// TIA Portal V17 export
// export: Created 2025-03-10T13:09:25.1133603Z, ExportSetting WithDefaults, DisplayName Totally Integrated Automation Portal, DisplayVersion V17 Update 8, DisplayName TIA Portal Openness, DisplayVersion V17 Update 8, DisplayName TIA Portal Version Control Interface, DisplayVersion V17, DisplayName SINAMICS Startdrive Advanced, DisplayVersion V17 SP2, DisplayName SINAMICS Startdrive G110M, G120, G120C, G120D, G120P, G115D, DisplayVersion V17 SP2, DisplayName SINAMICS Startdrive G130, G150, S120, S150, SINAMICS MV, S210, DisplayVersion V17 SP2, DisplayName STEP 7 Professional, DisplayVersion V17 Update 8, DisplayName SINUMERIK ONE STEP 7 Toolbox, DisplayVersion V17 Update 12, DisplayName SINUMERIK 840D sl STEP 7 Toolbox, DisplayVersion V17 Update 12, DisplayName STEP 7 Safety, DisplayVersion V17 Update 6, DisplayName WinCC Advanced, DisplayVersion V17 Update 8
DATA_BLOCK "LBP_PIServices"   // DB16
TITLE = PI Services / Servicios de IP / PI-Dienste
{ DB_Accessible_From_OPC_UA := 'FALSE' }
// Interface for LBP_ReqPIService [FB7], contains definitions for all available PI services. / Interfaz para LBP_ReqPIService [FB7], contiene definiciones para todos los servicios PI disponibles. / Schnittstelle für LBP_ReqPIService [FB7], enthält Definitionen für alle verfügbaren PI-Dienste.
// stored: DBAccessibleFromOPCUA false, DBAccessibleFromWebserver true, IsOnlyStoredInLoadMemory false, IsWriteProtectedInAS false
   VAR
      SELECT : Struct
         PIName : String[10] := '_N_SELECT';
         p01 : Byte := BYTE#16#03;   // Bereich/Einheit / Area / Unit / Área/unidad
         p02 : Char := '2';   // Bereichskennung / Area identifier / Identificador de área
         p11 : Byte := BYTE#16#FD;   // Pfad-Name / Path name / Nombre de ruta
         p12 : Byte := BYTE#16#13;   // String beliebig lang ungeradzahlig ergaenzen / Add string with arbitrary number of odd numbers / Completar string con cifras impares de una longitud cualquiera
         p21 : Byte := BYTE#16#FE;   // Programm-Name / Program name / Nombre de programa
         p22 : Byte := BYTE#16#13;   // String beliebig lang ungeradzahlig ergaenzen / Add string with arbitrary number of odd numbers / Completar string con cifras impares de una longitud cualquiera
      END_STRUCT;
      ASUP : Struct
         PIName : String[10] := '_N_ASUP__';
         p01 : Byte := BYTE#16#03;   // Bereich/Einheit / Area / Unit / Área/unidad
         p02 : Char := '2';   // Bereichskennung / Area identifier / Identificador de área
         p11 : Byte := BYTE#16#03;   // Interrupt-Nummer / Interrupt number / Número de interrupción
         p12 : Byte := BYTE#16#05;   // Int aus WORD-Spezifikation / Int from WORD specification / INT a partir de especificación WORD
         p21 : Byte := BYTE#16#03;   // Priorität / Priority / Prioridad
         p22 : Byte := BYTE#16#05;   // Int aus WORD-Spezifikation / Int from WORD specification / INT a partir de especificación WORD
         p31 : Byte := BYTE#16#01;   // Liftfast
         p32 : Byte := BYTE#16#05;   // Int aus WORD-Spezifikation / Int from WORD specification / INT a partir de especificación WORD
         p41 : Byte := BYTE#16#01;   // Blocksync / Sinc bloque
         p42 : Byte := BYTE#16#05;   // Int aus WORD-Spezifikation / Int from WORD specification / INT a partir de especificación WORD
         p51 : Byte := BYTE#16#FD;   // Pfad-Name / Path name / Nombre de ruta
         p52 : Byte := BYTE#16#13;   // String beliebig lang ungeradzahlig ergaenzen / Add string with arbitrary number of odd numbers / Completar string con cifras impares de una longitud cualquiera
         p61 : Byte := BYTE#16#FE;   // Programm-Name / Program name / Nombre de programa
         p62 : Byte := BYTE#16#13;   // String beliebig lang ungeradzahlig ergaenzen / Add string with arbitrary number of odd numbers / Completar string con cifras impares de una longitud cualquiera
      END_STRUCT;
      FINDBL : Struct
         PIName : String[10] := '_N_FINDBL';
         p01 : Byte := BYTE#16#03;   // Bereich/Einheit / Area / Unit / Área/unidad
         p02 : Char := '2';
         p11 : Byte := BYTE#16#01;   // Vorlaufmodus / Preprocessing mode / Modo de marcha previa
         p12 : Byte := BYTE#16#04;   // Word aus WORD-Spezifikation / Word from WORD specification / Word desde especificación WORD
      END_STRUCT;
      SETUFR : Struct
         PIName : String[10] := '_N_SETUFR';
         p01 : Byte := BYTE#16#03;   // Bereich/Einheit / Area / Unit / Área/unidad
         p02 : Char := '2';
      END_STRUCT;
      CANCEL : Struct
         PIName : String[10] := '_N_CANCEL';
         p01 : Byte := BYTE#16#03;   // Bereich/Einheit / Area / Unit / Área/unidad
         p02 : Char := '0';
      END_STRUCT;
      DELETO : Struct
         PIName : String[10] := '_N_DELETO';
         p01 : Byte := BYTE#16#03;   // Bereich/Einheit / Area / Unit / Área/unidad
         p02 : Char := '4';
         p11 : Byte := BYTE#16#05;   // T-Nummer / T number / N.º T
         p12 : Byte := BYTE#16#05;   // Int aus WORD-Spezifikation / Int from WORD specification / INT a partir de especificación WORD
      END_STRUCT;
      CREATO : Struct
         PIName : String[10] := '_N_CREATO';
         p01 : Byte := BYTE#16#03;   // Bereich/Einheit / Area / Unit / Área/unidad
         p02 : Char := '4';
         p11 : Byte := BYTE#16#05;   // T-Nummer / T number / N.º T
         p12 : Byte := BYTE#16#05;   // Int aus WORD-Spezifikation / Int from WORD specification / INT a partir de especificación WORD
      END_STRUCT;
      CREACE : Struct
         PIName : String[10] := '_N_CREACE';
         p01 : Byte := BYTE#16#03;   // Bereich/Einheit / Area / Unit / Área/unidad
         p02 : Char := '4';
         p11 : Byte := BYTE#16#05;   // T-Nummer / T number / N.º T
         p12 : Byte := BYTE#16#05;   // Int aus WORD-Spezifikation / Int from WORD specification / INT a partir de especificación WORD
      END_STRUCT;
      TMCRTO : Struct
         PIName : String[10] := '_N_TMCRTO';
         p01 : Byte := BYTE#16#03;   // Bereich/Einheit / Area / Unit / Área/unidad
         p02 : Char := '4';
         p11 : Byte := BYTE#16#20;   // Werkzeugkennung, Leerzeichen hinzufügen / Tool identifier, add blank / Identificador de herramienta, agregar espacio en blanco
         p12 : Byte := BYTE#16#13;   // Stringkennung! / String identifier! / ¡Identificador de string!
         p21 : Byte := BYTE#16#05;   // T-Nummer / T number / N.º T
         p22 : Byte := BYTE#16#05;   // Int aus WORD-Spezifikation / Int from WORD specification / INT a partir de especificación WORD
         p31 : Byte := BYTE#16#05;   // Duplo Nummer / Duplo number / Número duplo
         p32 : Byte := BYTE#16#05;   // Int aus WORD-Spezifikation / Int from WORD specification / INT a partir de especificación WORD
      END_STRUCT;
      TMFDPL : Struct
         PIName : String[10] := '_N_TMFDPL';
         p01 : Byte := BYTE#16#03;   // Bereich/Einheit / Area / Unit / Área/unidad
         p02 : Char := '4';
         p11 : Byte := BYTE#16#05;   // T-Nummer / T number / N.º T
         p12 : Byte := BYTE#16#05;   // Int aus WORD-Spezifikation / Int from WORD specification / INT a partir de especificación WORD
         p21 : Byte := BYTE#16#05;   // Platznummer (Ziel) / Location number (target) / Número de puesto (destino)
         p22 : Byte := BYTE#16#05;   // Int aus WORD-Spezifikation / Int from WORD specification / INT a partir de especificación WORD
         p31 : Byte := BYTE#16#05;   // Magazinnummer (Ziel) / Magazine number (target) / Número de almacén (destino)
         p32 : Byte := BYTE#16#05;   // Int aus WORD-Spezifikation / Int from WORD specification / INT a partir de especificación WORD
         p41 : Byte := BYTE#16#05;   // Platznummer (Bezug) / Location number (reference) / Número de puesto (referencia)
         p42 : Byte := BYTE#16#05;   // Int aus WORD-Spezifikation / Int from WORD specification / INT a partir de especificación WORD
         p51 : Byte := BYTE#16#05;   // Magazin-Nummer (Bezug) / Magazine number (reference) / Número de almacén (referencia)
         p52 : Byte := BYTE#16#05;   // Int aus WORD-Spezifikation / Int from WORD specification / INT a partir de especificación WORD
      END_STRUCT;
      TMMVTL : Struct
         PIName : String[10] := '_N_TMMVTL';
         p01 : Byte := BYTE#16#03;   // Bereich/Einheit / Area / Unit / Área/unidad
         p02 : Char := '4';
         p11 : Byte := BYTE#16#05;   // T-Nummer / T number / N.º T
         p12 : Byte := BYTE#16#05;   // Int aus WORD-Spezifikation / Int from WORD specification / INT a partir de especificación WORD
         p21 : Byte := BYTE#16#05;   // Platznummer (Quelle) / Location number (source) / Número de puesto (origen)
         p22 : Byte := BYTE#16#05;   // Int aus WORD-Spezifikation / Int from WORD specification / INT a partir de especificación WORD
         p31 : Byte := BYTE#16#05;   // Magazin-Nummer (Quelle) / Magazine number (source) / Número de almacén (origen)
         p32 : Byte := BYTE#16#05;   // Int aus WORD-Spezifikation / Int from WORD specification / INT a partir de especificación WORD
         p41 : Byte := BYTE#16#05;   // Platznummer (Ziel) / Location number (target) / Número de puesto (destino)
         p42 : Byte := BYTE#16#05;   // Int aus WORD-Spezifikation / Int from WORD specification / INT a partir de especificación WORD
         p51 : Byte := BYTE#16#05;   // Magazin-Nummer (Ziel) / Magazine number (target) / Número de almacén (destino)
         p52 : Byte := BYTE#16#05;   // Int aus WORD-Spezifikation / Int from WORD specification / INT a partir de especificación WORD
      END_STRUCT;
      TMPCIT : Struct
         PIName : String[10] := '_N_TMPCIT';
         p01 : Byte := BYTE#16#03;   // Bereich/Einheit / Area / Unit / Área/unidad
         p02 : Char := '4';
         p11 : Byte := BYTE#16#03;   // Spindelnummer / Spindle number / Número de cabezal
         p12 : Byte := BYTE#16#05;   // Int aus WORD-Spezifikation / Int from WORD specification / INT a partir de especificación WORD
         p21 : Byte := BYTE#16#05;   // Inkrement Wert / Increment value / Valor incremental
         p22 : Byte := BYTE#16#05;   // Int aus WORD-Spezifikation / Int from WORD specification / INT a partir de especificación WORD
      END_STRUCT;
      TMPOSM : Struct
         PIName : String[10] := '_N_TMPOSM';
         p01 : Byte := BYTE#16#03;   // Bereich/Einheit / Area / Unit / Área/unidad
         p02 : Char := '4';
         p11 : Byte := BYTE#16#05;   // T-Nummer / T number / N.º T
         p12 : Byte := BYTE#16#05;   // Int aus WORD-Spezifikation / Int from WORD specification / INT a partir de especificación WORD
         p21 : Byte := BYTE#16#20;   // Werkzeugbezeichner, Leerzeichen hinzufügen / Tool identifier, add blank / Identificador de herramienta, agregar espacio en blanco
         p22 : Byte := BYTE#16#13;   // Stringkennung! / String identifier! / ¡Identificador de string!
         p31 : Byte := BYTE#16#05;   // Duplo Nummer / Duplo number / Número duplo
         p32 : Byte := BYTE#16#05;   // Int aus WORD-Spezifikation / Int from WORD specification / INT a partir de especificación WORD
         p41 : Byte := BYTE#16#05;   // Platznummer (Quelle) / Location number (source) / Número de puesto (origen)
         p42 : Byte := BYTE#16#05;   // Int aus WORD-Spezifikation / Int from WORD specification / INT a partir de especificación WORD
         p51 : Byte := BYTE#16#05;   // Magazin-Nummer (Quelle) / Magazine number (source) / Número de almacén (origen)
         p52 : Byte := BYTE#16#05;   // Int aus WORD-Spezifikation / Int from WORD specification / INT a partir de especificación WORD
         p61 : Byte := BYTE#16#05;   // Platznummer (Ziel) / Location number (target) / Número de puesto (destino)
         p62 : Byte := BYTE#16#05;   // Int aus WORD-Spezifikation / Int from WORD specification / INT a partir de especificación WORD
         p71 : Byte := BYTE#16#05;   // Magazin-Nummer (Ziel) / Magazine number (target) / Número de almacén (destino)
         p72 : Byte := BYTE#16#05;   // Int aus WORD-Spezifikation / Int from WORD specification / INT a partir de especificación WORD
      END_STRUCT;
      DIGION : Struct
         PIName : String[10] := '_N_DIGION';
         p01 : Byte := BYTE#16#03;   // Bereich/Einheit / Area / Unit / Área/unidad
         p02 : Char := '2';
      END_STRUCT;
      DIGIOF : Struct
         PIName : String[10] := '_N_DIGIOF';
         p01 : Byte := BYTE#16#03;   // Bereich/Einheit / Area / Unit / Área/unidad
         p02 : Char := '2';
      END_STRUCT;
      CONFIG : Struct
         PIName : String[10] := '_N_CONFIG';
         p01 : Byte := BYTE#16#03;   // Bereich/Einheit / Area / Unit / Área/unidad
         p02 : Char := '0';
         p11 : Byte := BYTE#16#02;   // Klassifizierung / Classification / Clasificación
         p12 : Byte := BYTE#16#04;   // Int aus WORD-Spezifikation / Int from WORD specification / INT a partir de especificación WORD
      END_STRUCT;
      LOGIN : Struct
         PIName : String[10] := '_N_LOGIN_';
         p01 : Byte := BYTE#16#03;   // Bereich/Einheit / Area / Unit / Área/unidad
         p02 : Char := '0';
         p11 : Byte := BYTE#16#20;   // Kennwort (8 - 32 Zeichen) / Password (8 to 32 characters) / Contraseña (de 8 a 32 caracteres)
         p12 : Byte := BYTE#16#13;   // Stringkennung! / String identifier! / ¡Identificador de string!
      END_STRUCT;
      LOGOUT : Struct
         PIName : String[10] := '_N_LOGOUT';
         p01 : Byte := BYTE#16#03;   // Bereich/Einheit / Area / Unit / Área/unidad
         p02 : Char := '0';
      END_STRUCT;
      MMCSEM : Struct
         PIName : String[10] := '_N_MMCSEM';
         p01 : Byte := BYTE#16#03;   // Bereich/Einheit / Area / Unit / Área/unidad
         p02 : Char := '2';
         p11 : Byte := BYTE#16#03;   // Funktionsnummer / Function number / Número de función
         p12 : Byte := BYTE#16#05;   // Int aus WORD-Spezifikation / Int from WORD specification / INT a partir de especificación WORD
         p21 : Byte := BYTE#16#01;   // Semaphore-Wert / Semaphore value / Valor de semáforo
         p22 : Byte := BYTE#16#05;   // Int aus WORD-Spezifikation / Int from WORD specification / INT a partir de especificación WORD
      END_STRUCT;
      DELECE : Struct
         PIName : String[10] := '_N_DELECE';
         p01 : Byte := BYTE#16#03;   // Bereich/Einheit / Area / Unit / Área/unidad
         p02 : Char := '4';
         p11 : Byte := BYTE#16#05;   // T-Nummer / T number / N.º T
         p12 : Byte := BYTE#16#05;   // Int aus WORD-Spezifikation / Int from WORD specification / INT a partir de especificación WORD
         p21 : Byte := BYTE#16#05;   // D-Nummer / D number / N.º D
         p22 : Byte := BYTE#16#05;   // Int aus WORD-Spezifikation / Int from WORD specification / INT a partir de especificación WORD
      END_STRUCT;
      CRCEDN : Struct
         PIName : String[10] := '_N_CRCEDN';
         p01 : Byte := BYTE#16#03;   // Bereich/Einheit / Area / Unit / Área/unidad
         p02 : Char := '4';
         p11 : Byte := BYTE#16#05;   // T-Nummer / T number / N.º T
         p12 : Byte := BYTE#16#05;   // Int aus WORD-Spezifikation / Int from WORD specification / INT a partir de especificación WORD
         p21 : Byte := BYTE#16#05;   // D-Nummer / D number / N.º D
         p22 : Byte := BYTE#16#05;   // Int aus WORD-Spezifikation / Int from WORD specification / INT a partir de especificación WORD
      END_STRUCT;
      TSEARC : Struct
         PIName : String[10] := '_N_TSEARC';
         p01 : Byte := BYTE#16#03;   // Bereich/Einheit / Area / Unit / Área/unidad
         p02 : Char := '4';
         p11 : Byte := BYTE#16#05;   // von: Magazin-Nummer / from: Magazine number / desde: número de almacén
         p12 : Byte := BYTE#16#05;   // Int aus WORD-Spezifikation / Int from WORD specification / INT a partir de especificación WORD
         p21 : Byte := BYTE#16#05;   // von: Platznummer / from: Location number / desde: número de puesto
         p22 : Byte := BYTE#16#05;   // Int aus WORD-Spezifikation / Int from WORD specification / INT a partir de especificación WORD
         p31 : Byte := BYTE#16#05;   // bis: Magazin-Nummer / up to: Magazine number / hasta: número de almacén
         p32 : Byte := BYTE#16#05;   // Int aus WORD-Spezifikation / Int from WORD specification / INT a partir de especificación WORD
         p41 : Byte := BYTE#16#05;   // bis: Platznummer / up to: Location number / hasta: número de puesto
         p42 : Byte := BYTE#16#05;   // Int aus WORD-Spezifikation / Int from WORD specification / INT a partir de especificación WORD
         p51 : Byte := BYTE#16#05;   // Nummer des Referenz-Magazins / Number of reference magazine / Número del almacén de referencia
         p52 : Byte := BYTE#16#05;   // Int aus WORD-Spezifikation / Int from WORD specification / INT a partir de especificación WORD
         p61 : Byte := BYTE#16#05;   // Nummer des Referenz-Platzes / Number of reference location / Número del puesto de referencia
         p62 : Byte := BYTE#16#05;   // Int aus WORD-Spezifikation / Int from WORD specification / INT a partir de especificación WORD
         p71 : Byte := BYTE#16#01;   // Suchrichtung / Search direction / Sentido de búsqueda
         p72 : Byte := BYTE#16#05;   // Int aus WORD-Spezifikation / Int from WORD specification / INT a partir de especificación WORD
         p81 : Byte := BYTE#16#01;   // Eigenschaften der Werkzeuge / Tool properties / Propiedades de las herramientas
         p82 : Byte := BYTE#16#05;   // Int aus WORD-Spezifikation / Int from WORD specification / INT a partir de especificación WORD
      END_STRUCT;
      TMFPBP : Struct
         PIName : String[10] := '_N_TMFPBP';
         p01 : Byte := BYTE#16#03;   // Bereich/Einheit / Area / Unit / Área/unidad
         p02 : Char := '4';
         p11 : Byte := BYTE#16#05;   // von: Magazin-Nummer / from: Magazine number / desde: número de almacén
         p12 : Byte := BYTE#16#05;   // Int aus WORD-Spezifikation / Int from WORD specification / INT a partir de especificación WORD
         p21 : Byte := BYTE#16#05;   // von: Platznummer / from: Location number / desde: número de puesto
         p22 : Byte := BYTE#16#05;   // Int aus WORD-Spezifikation / Int from WORD specification / INT a partir de especificación WORD
         p31 : Byte := BYTE#16#05;   // bis: Magazin Nummer / up to: Magazine number / hasta: número de almacén
         p32 : Byte := BYTE#16#05;   // Int aus WORD-Spezifikation / Int from WORD specification / INT a partir de especificación WORD
         p41 : Byte := BYTE#16#05;   // bis: Platznummer / up to: Location number / hasta: número de puesto
         p42 : Byte := BYTE#16#05;   // Int aus WORD-Spezifikation / Int from WORD specification / INT a partir de especificación WORD
         p51 : Byte := BYTE#16#05;   // Nummer des Referenz-Magazins / Number of reference magazine / Número del almacén de referencia
         p52 : Byte := BYTE#16#05;   // Int aus WORD-Spezifikation / Int from WORD specification / INT a partir de especificación WORD
         p61 : Byte := BYTE#16#05;   // Nummer des Referenz-Platzes / Number of reference location / Número del puesto de referencia
         p62 : Byte := BYTE#16#05;   // Int aus WORD-Spezifikation / Int from WORD specification / INT a partir de especificación WORD
         p71 : Byte := BYTE#16#05;   // Anzahl der Plätze nach links / Number of locations to the left / Número de puestos hacia la izquierda
         p72 : Byte := BYTE#16#05;   // Int aus WORD-Spezifikation / Int from WORD specification / INT a partir de especificación WORD
         p81 : Byte := BYTE#16#05;   // Anzahl der Plätze nach rechts / Number of locations to the right / Número de puestos hacia la derecha
         p82 : Byte := BYTE#16#05;   // Int aus WORD-Spezifikation / Int from WORD specification / INT a partir de especificación WORD
         p91 { ExternalVisible := 'False'} : Byte := BYTE#16#05;   // Anzahl der Plätze nach oben / Number of locations above / Número de puestos hacia arriba
         p92 : Byte := BYTE#16#05;   // Int aus WORD-Spezifikation / Int from WORD specification / INT a partir de especificación WORD
         pa1 : Byte := BYTE#16#05;   // Anzahl der Plätze nach unten / Number of locations below / Número de puestos hacia abajo
         pa2 : Byte := BYTE#16#05;   // Int aus WORD-Spezifikation / Int from WORD specification / INT a partir de especificación WORD
         pb1 : Byte := BYTE#16#05;   // Platztyp Index / Location type index / Índice tipo de puesto
         pb2 : Byte := BYTE#16#05;   // Int aus WORD-Spezifikation / Int from WORD specification / INT a partir de especificación WORD
         pc1 : Byte := BYTE#16#05;   // Suchrichtung / Search direction / Sentido de búsqueda
         pc2 : Byte := BYTE#16#05;   // Int aus WORD-Spezifikation / Int from WORD specification / INT a partir de especificación WORD
      END_STRUCT;
      NCRES : Struct
         PIName : String[10] := '_N_IBN_SS';
         p01 : Byte := BYTE#16#03;   // Bereich/Einheit / Area / Unit / Área/unidad
         p02 : Char := 'K';
         p11 : Byte := BYTE#16#01;   // Klassifizierung / Classification / Clasificación
         p12 : Byte := BYTE#16#04;   // WORD-Spezifikation / WORD specification / Especificación WORD
      END_STRUCT;
      TMRASS : Struct
         PIName : String[10] := '_N_TMRASS';
         p01 : Byte := BYTE#16#03;   // Bereich/Einheit / Area / Unit / Área/unidad
         p02 : Char := '4';
      END_STRUCT;
      TRESMO : Struct
         PIName : String[10] := '_N_TRESMO';
         p01 : Byte := BYTE#16#03;   // Bereich/Einheit / Area / Unit / Área/unidad
         p02 : Char := '4';
         p11 : Byte := BYTE#16#05;   // Werkzeugnummer / Tool number / Número de herramienta
         p12 : Byte := BYTE#16#05;   // Int aus WORD-Spezifikation / Int from WORD specification / INT a partir de especificación WORD
         p21 : Byte := BYTE#16#05;   // D-Nummer / D number / N.º D
         p22 : Byte := BYTE#16#05;   // Int aus WORD-Spezifikation / Int from WORD specification / INT a partir de especificación WORD
         p31 : Byte := BYTE#16#05;   // Überwachungsart / Monitoring type / Tipo de vigilancia
         p32 : Byte := BYTE#16#05;   // Int aus WORD-Spezifikation / Int from WORD specification / INT a partir de especificación WORD
      END_STRUCT;
      TMGETT : Struct
         PIName : String[10] := '_N_TMGETT';
         p01 : Byte := BYTE#16#03;   // Bereich/Einheit / Area / Unit / Área/unidad
         p02 : Char := '4';
         p11 : Byte := BYTE#16#20;   // Werkzeugkennung, Leerzeichen hinzufügen / Tool identifier, add blank / Identificador de herramienta, agregar espacio en blanco
         p12 : Byte := BYTE#16#13;   // Stringkennung! / String identifier! / ¡Identificador de string!
         p21 : Byte := BYTE#16#05;   // Duplonummer / Duplo number / Número duplo
         p22 : Byte := BYTE#16#05;   // Int aus WORD-Spezifikation / Int from WORD specification / INT a partir de especificación WORD
      END_STRUCT;
      SETUDT : Struct
         PIName : String[10] := '_N_SETUDT';
         p01 : Byte := BYTE#16#03;   // Bereich/Einheit / Area / Unit / Área/unidad
         p02 : Char := '2';
         p11 : Byte := BYTE#16#03;   // UserDataType
         p12 : Byte := BYTE#16#04;   // WORD-Spezifikation / WORD specification / Especificación WORD
         p21 : Byte := BYTE#16#05;   // ind1
         p22 : Byte := BYTE#16#04;   // WORD-Spezifikation / WORD specification / Especificación WORD
         p31 : Byte := BYTE#16#05;   // ind2
         p32 : Byte := BYTE#16#04;   // WORD-Spezifikation / WORD specification / Especificación WORD
      END_STRUCT;
      TMCRMT : Struct
         PIName : String[10] := '_N_TMCRMT';
         p01 : Byte := BYTE#16#03;   // Bereich/Einheit / Area / Unit / Área/unidad
         p02 : Char := '4';
         p11 : Byte := BYTE#16#20;   // Multitool-Bezeichner, Leerzeichen einfügen / Multitool identifier, insert blanks / Identificador Multitool, agregar espacio en blanco
         p12 : Byte := BYTE#16#13;   // Stringkennung! / String identifier! / ¡Identificador de string!
         p21 : Byte := BYTE#16#05;   // Reserviert / Reserved / Reservado
         p22 : Byte := BYTE#16#05;   // Int aus WORD-Spezifikation / Int from WORD specification / INT a partir de especificación WORD
         p31 : Byte := BYTE#16#05;   // Multitool-Nummer / Multitool number / Número de Multitool
         p32 : Byte := BYTE#16#05;   // Int aus WORD-Spezifikation / Int from WORD specification / INT a partir de especificación WORD
         p41 : Byte := BYTE#16#03;   // Anzahl der Plätze im Multitool / Number of Multitool locations / Número de puestos en Multitool
         p42 : Byte := BYTE#16#05;   // Int aus WORD-Spezifikation / Int from WORD specification / INT a partir de especificación WORD
         p51 : Byte := BYTE#16#01;   // Art der Abstandskodierung / Type of distance coding / Tipo de codificación de distancia
         p52 : Byte := BYTE#16#05;   // Int aus WORD-Spezifikation / Int from WORD specification / INT a partir de especificación WORD
      END_STRUCT;
      TMDLMT : Struct
         PIName : String[10] := '_N_TMDLMT';
         p01 : Byte := BYTE#16#03;   // Bereich/Einheit / Area / Unit / Área/unidad
         p02 : Char := '4';
         p11 : Byte := BYTE#16#20;   // Multitool-Bezeichner, Leerzeichen einfügen / Multitool identifier, insert blanks / Identificador Multitool, agregar espacio en blanco
         p12 : Byte := BYTE#16#13;   // Stringkennung! / String identifier! / ¡Identificador de string!
         p21 : Byte := BYTE#16#05;   // Reserviert / Reserved / Reservado
         p22 : Byte := BYTE#16#05;   // Int aus WORD-Spezifikation / Int from WORD specification / INT a partir de especificación WORD
         p31 : Byte := BYTE#16#05;   // Multitool-Nummer / Multitool number / Número de Multitool
         p32 : Byte := BYTE#16#05;   // Int aus WORD-Spezifikation / Int from WORD specification / INT a partir de especificación WORD
         p41 : Byte := BYTE#16#01;   // Lösche enthaltene Werkzeuge / Delete included tools / Borrar herramientas incluidas
         p42 : Byte := BYTE#16#05;   // Int aus WORD-Spezifikation / Int from WORD specification / INT a partir de especificación WORD
      END_STRUCT;
      POSMT : Struct
         PIName : String[10] := '_N_POSMT_';
         p01 : Byte := BYTE#16#03;   // Bereich/Einheit / Area / Unit / Área/unidad
         p02 : Char := '4';
         p11 : Byte := BYTE#16#03;   // Nummer des Werkzeughalters / Number of toolholder / Número del portaherramientas
         p12 : Byte := BYTE#16#05;   // Int aus WORD-Spezifikation / Int from WORD specification / INT a partir de especificación WORD
         p21 : Byte := BYTE#16#05;   // Werkzeugnummer / Tool number / Número de herramienta
         p22 : Byte := BYTE#16#05;   // Int aus WORD-Spezifikation / Int from WORD specification / INT a partir de especificación WORD
         p31 : Byte := BYTE#16#20;   // Werkzeugnummer, Leerzeichen hinzufügen / Tool number, add blank / Número de herramienta, agregar espacio en blanco
         p32 : Byte := BYTE#16#13;   // Stringkennung! / String identifier! / ¡Identificador de string!
         p41 : Byte := BYTE#16#05;   // Duplonummer / Duplo number / Número duplo
         p42 : Byte := BYTE#16#05;   // Int aus WORD-Spezifikation / Int from WORD specification / INT a partir de especificación WORD
         p51 : Byte := BYTE#16#03;   // Multitool-Platznummer / Multitool place number / Número de puesto de Multitool
         p52 : Byte := BYTE#16#05;   // Int aus WORD-Spezifikation / Int from WORD specification / INT a partir de especificación WORD
      END_STRUCT;
      FDPLMT : Struct
         PIName : String[10] := '_N_FDPLMT';
         p01 : Byte := BYTE#16#03;   // Bereich/Einheit / Area / Unit / Área/unidad
         p02 : Char := '4';
         p11 : Byte := BYTE#16#05;   // Werkzeugnummer / Tool number / Número de herramienta
         p12 : Byte := BYTE#16#05;   // Int aus WORD-Spezifikation / Int from WORD specification / INT a partir de especificación WORD
         p21 : Byte := BYTE#16#20;   // Werkzeugnummer, Leerzeichen hinzufügen / Tool number, add blank / Número de herramienta, agregar espacio en blanco
         p22 : Byte := BYTE#16#13;   // Stringkennung! / String identifier! / ¡Identificador de string!
         p31 : Byte := BYTE#16#05;   // Duplonummer / Duplo number / Número duplo
         p32 : Byte := BYTE#16#05;   // Int aus WORD-Spezifikation / Int from WORD specification / INT a partir de especificación WORD
         p41 : Byte := BYTE#16#05;   // Multitool-Nummer / Multitool number / Número de Multitool
         p42 : Byte := BYTE#16#05;   // Int aus WORD-Spezifikation / Int from WORD specification / INT a partir de especificación WORD
         p51 : Byte := BYTE#16#03;   // Multitool-Platznummer / Multitool place number / Número de puesto de Multitool
         p52 : Byte := BYTE#16#05;   // Int aus WORD-Spezifikation / Int from WORD specification / INT a partir de especificación WORD
      END_STRUCT;
      RETRAC : Struct
         PIName : String[10] := '_N_RETRAC';
         p01 : Byte := BYTE#16#03;   // Bereich/Einheit / Area / Unit / Área/unidad
         p02 : Char := '2';
         p11 : Byte := BYTE#16#03;   // Geometrieachse / Geometry axis / Eje geométrico
         p12 : Byte := BYTE#16#04;   // WORD-Spezifikation / WORD specification / Especificación WORD
         p21 : Byte := BYTE#16#05;   // Parameter2 / Parámetro2
         p22 : Byte := BYTE#16#04;   // WORD-Spezifikation / WORD specification / Especificación WORD
      END_STRUCT;
   END_VAR
BEGIN
END_DATA_BLOCK
